FUNCTION_BLOCK Frequency_Power (* Composite Function Block Type *)
  (* Standard: 61499-2 *)
  (* Version 0.0, 7/5/2024, SESA371406, Schneider Electric, template *)
  PACKAGE SE.Nereda;
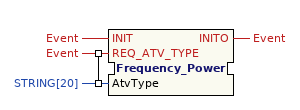
  EVENT_INPUT
    INIT; (* Initializes the symbolic link data destination FB with N (1 <= N <= 16) variables *)
    REQ_ATV_TYPE WITH AtvType;
  END_EVENT
  EVENT_OUTPUT
    INITO;
  END_EVENT
  VAR_INPUT
    AtvType : STRING[20];
  END_VAR
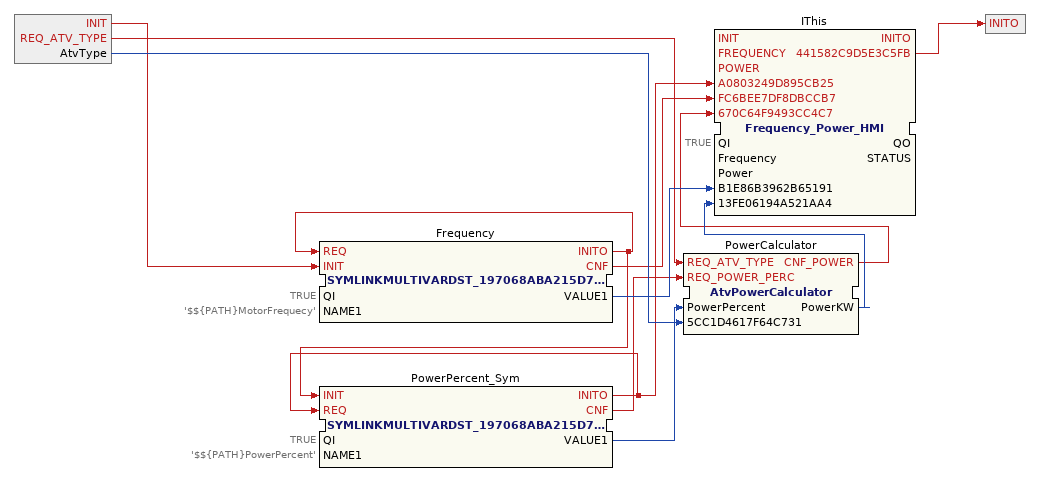
  (* 01 - FUNCTIONNAL INPUT INTERFACE *)
  (* 00 - INITIALIZATION *)
  (* 05 - LOGIC *)
  (* 06 - HMI INTERFACE *)
  (* 03 - FIELD INTERFACE *)
  (* 02 - FUNCTIONNAL OUTPUT INTERFACE *)
  (* Power Calculator *)
  FBS
    IThis : Frequency_Power_HMI(QI := TRUE);
    Frequency : SYMLINKMULTIVARDST_197068ABA215D7EBA(QI := TRUE, NAME1 := '$${PATH}MotorFrequecy'); {SET_ATTRIBUTE(Configuration.GenericFBType.InterfaceParams, Runtime.System#I:=1;VALUE${I$}:REAL)}
    PowerPercent_Sym : SYMLINKMULTIVARDST_197068ABA215D7EBA(QI := TRUE, NAME1 := '$${PATH}PowerPercent'); {SET_ATTRIBUTE(Configuration.GenericFBType.InterfaceParams, Runtime.System#I:=1;VALUE${I$}:REAL)}
    PowerCalculator : AtvPowerCalculator;
  END_FBS
  EVENT_CONNECTIONS
    Frequency.INITO TO PowerPercent_Sym.INIT;
    Frequency.INITO TO Frequency.REQ;
    PowerPercent_Sym.INITO TO PowerPercent_Sym.REQ;
    INIT TO Frequency.INIT;
    PowerPercent_Sym.INITO TO IThis.A0803249D895CB25;
    Frequency.CNF TO IThis.FC6BEE7DF8DBCCB7;
    IThis.441582C9D5E3C5FB TO INITO;
    REQ_ATV_TYPE TO PowerCalculator.REQ_ATV_TYPE;
    PowerPercent_Sym.CNF TO PowerCalculator.REQ_POWER_PERC;
    PowerCalculator.CNF_POWER TO IThis.670C64F9493CC4C7;
  END_CONNECTIONS
  DATA_CONNECTIONS
    Frequency.VALUE1 TO IThis.B1E86B3962B65191;
    PowerPercent_Sym.VALUE1 TO PowerCalculator.PowerPercent;
    AtvType TO PowerCalculator.5CC1D4617F64C731;
    PowerCalculator.PowerKW TO IThis.13FE06194A521AA4;
  END_CONNECTIONS
END_FUNCTION_BLOCK
